// TIA Portal V18 export
ORGANIZATION_BLOCK "AutoLogic"   // OB1, FBD, ProgramCycle
TITLE = "Main Program Sweep (Cycle)"
{ S7_Optimized_Access := 'TRUE' }
VERSION : 0.1
// stored: AutoNumber true, IsIECCheckEnabled false, SetENOAutomatically false
   VAR_INPUT
      Initial_Call : Bool;   // Initial call of this OB
      Remanence : Bool;   // =True, if remanent data are available
   END_VAR
   VAR_TEMP
      UTL_TIME : Array[0..2] of DInt;
      chbs_cmd : Bool;
      chbr_cmd : Bool;
      STEAM_MAN_SCV_MVE : Real;
      STEAM_SCV_MVE : Real;
      STEAM_SCV_SCL : Real;
   END_VAR
BEGIN

REGION Network 1: Source select
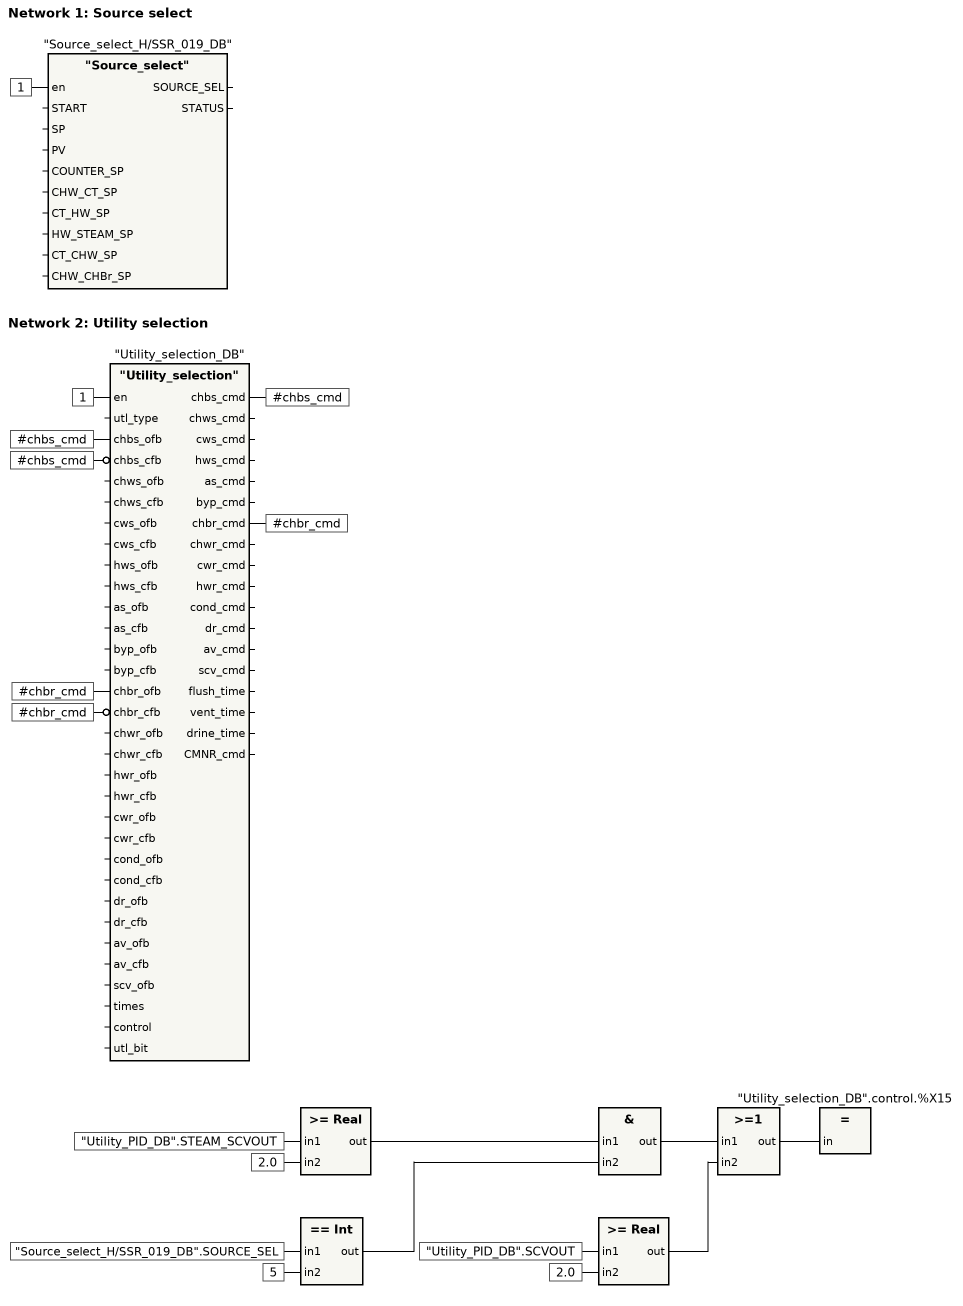
   IF 1 THEN
       "Source_select_H/SSR_019_DB"();   // "Source_select"
   END_IF;
END_REGION

REGION Network 2: Utility selection
   IF 1 THEN
       "Utility_selection_DB"(chbs_ofb := #chbs_cmd,   // "Utility_selection"
                              chbs_cfb := NOT #chbs_cmd,
                              chbr_ofb := #chbr_cmd,
                              chbr_cfb := NOT #chbr_cmd,
                              chbs_cmd => #chbs_cmd,
                              chbr_cmd => #chbr_cmd);
   END_IF;
   "Utility_selection_DB".control.%X15 := (("Utility_PID_DB".STEAM_SCVOUT >= 2.0) AND ("Source_select_H/SSR_019_DB".SOURCE_SEL = 5)) OR ("Utility_PID_DB".SCVOUT >= 2.0);
END_REGION
END_ORGANIZATION_BLOCK
